# EPICS substitutions: db/Baumer/ecmcEAx580.substitutions
file "ecmcEAx580-chX.template"
{
  pattern {CH_ID}
          {01   }
}
